{attribute 'GeneratedUsingTerminal: EL3356-0030-0025'}
{attribute addProperty BoxType "EL3356-0030-0025"}
{attribute addProperty Id "EtcSlaveTerminalBaseRMB_StatusAT %I*RMB_Status_C0E100AA7RMB_Value_INT32AT %I*RMB_Value_INT_E9189C4B4RMB_ControlAT %Q*RMB_Control_CC49845C5WcStateAT %I*WcState_9091E0EB2InfoDataAT %I*InfoData_32EB74EA10"}
{attribute addProperty CRC "3201882295"}
{attribute addProperty Size "28"}
TYPE EL3356_BED8D8B7 EXTENDS EtcSlaveTerminalBase :
STRUCT
	{attribute addProperty Name "RMB_Status"}
	RMB_Status : RMB_Status_C0E100AA;
	{attribute addProperty Name "RMB_Value_INT32"}
	RMB_Value_INT32 : RMB_Value_INT_E9189C4B;
	{attribute addProperty Name "RMB_Control"}
	RMB_Control : RMB_Control_CC49845C;
	{attribute addProperty Name "WcState"}
	WcState : WcState_9091E0EB;
	{attribute addProperty Name "InfoData"}
	InfoData : InfoData_32EB74EA;
END_STRUCT
END_TYPE

(* stored: Version 1.2.0.0, ProductVersion 3.1.4024.9
   DUT EL3356_BED8D8B7: Id {0caa7926-ac63-4eae-87c3-d98f1208323d} *)
